# EPICS substitutions: db/Beckhoff_1XXX/ecmcEL1252.substitutions
file "ecmcEcSlave.template"
{
  pattern {}
          {}
}

file "ecmcEX1XXX.template"
{
  pattern {CH_ID, ZNAM,   ONAM,   ZSV,        OSV,        PINI,  DESC                              }
          {1,     "Zero", "One",  "NO_ALARM", "NO_ALARM", 1,     "$(HWTYPE): Binary Input $(CH_ID)"}
          {2,     "Zero", "One",  "NO_ALARM", "NO_ALARM", 1,     "$(HWTYPE): Binary Input $(CH_ID)"}
}

# Timestamps and status words
file "ecmcEL1252.template"
{
  pattern {CH_ID, PINI }
          {1,     1    }
          {2,     1    }
}
